{attribute 'GeneratedUsingTerminal: EP6224-0002-0016'}
{attribute addProperty BoxType "EP6224-0002-0016"}
{attribute addProperty Id "Digital_InputsDigital_Inputs_FE0422394"}
{attribute addProperty CRC "4069995187"}
{attribute addProperty Size "4"}
TYPE Module_7_Digital_Inputs_F29732B3 :
STRUCT
	{attribute addProperty Name "Digital_Inputs"}
	Digital_Inputs  : Digital_Inputs_FE042239;
END_STRUCT
END_TYPE

(* stored: Version 1.2.0.0, ProductVersion 3.1.4024.9
   DUT Module_7_Digital_Inputs_F29732B3: Id {23fe7e1d-27fd-4d41-a4ba-fe21dcfb37c3} *)
